FUNCTION_BLOCK TcoContextEnvironment IMPLEMENTS ITcoContextEnvironment
VAR
	_messenger : TcoMessengerSettings;
END_VAR

(*~
		<docu>
			<summary>
				Gets messaging settings of this context.			
			</summary>			
		</docu>	
~*)
PROPERTY Messaging : ITcoMessengerSettings
GET
Messaging := _messenger;
END_GET
END_PROPERTY

END_FUNCTION_BLOCK

(* stored: Version 1.1.0.1, ProductVersion 3.1.4024.9
   POU TcoContextEnvironment: Id {3220df02-9b69-0aaa-1c5f-41ed13d5599f}, SpecialFunc None
   Property Messaging: Id {80bc198f-e53b-04f5-1cbc-ef3a2ee37c8f}
   Get Get: Id {2afecb4e-9dba-0868-0a02-c655cbf5e0a9} *)
